FUNCTION_BLOCK UNIT_StateLogic (* Reduced PackML unit state machine: Reset/Start/Clear only from the occupation owner and only in a valid state; Execute runs the procedure until it reports DONE (Complete) or FAILED (Aborted) *)
  (* Standard: 61499-2 *)
  (* Version 0.1, 2026-09-28, Project contributors, AAU Smart Production Lab *)
  PACKAGE unitlib;
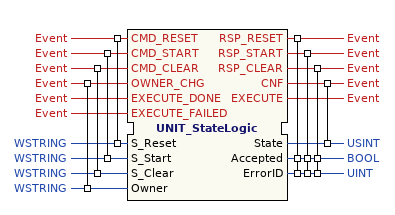
  EVENT_INPUT
    CMD_RESET WITH S_Reset;
    CMD_START WITH S_Start;
    CMD_CLEAR WITH S_Clear;
    OWNER_CHG WITH Owner;
    EXECUTE_DONE;
    EXECUTE_FAILED;
  END_EVENT
  EVENT_OUTPUT
    RSP_RESET WITH Accepted, ErrorID;
    RSP_START WITH Accepted, ErrorID;
    RSP_CLEAR WITH Accepted, ErrorID;
    CNF WITH State;
    EXECUTE;
  END_EVENT
  VAR_INPUT
    S_Reset : WSTRING;
    S_Start : WSTRING;
    S_Clear : WSTRING;
    Owner : WSTRING;
  END_VAR
  VAR_OUTPUT
    State : USINT := 2;
    Accepted : BOOL;
    ErrorID : UINT;
  END_VAR
  VAR
    Owned : BOOL;
  END_VAR
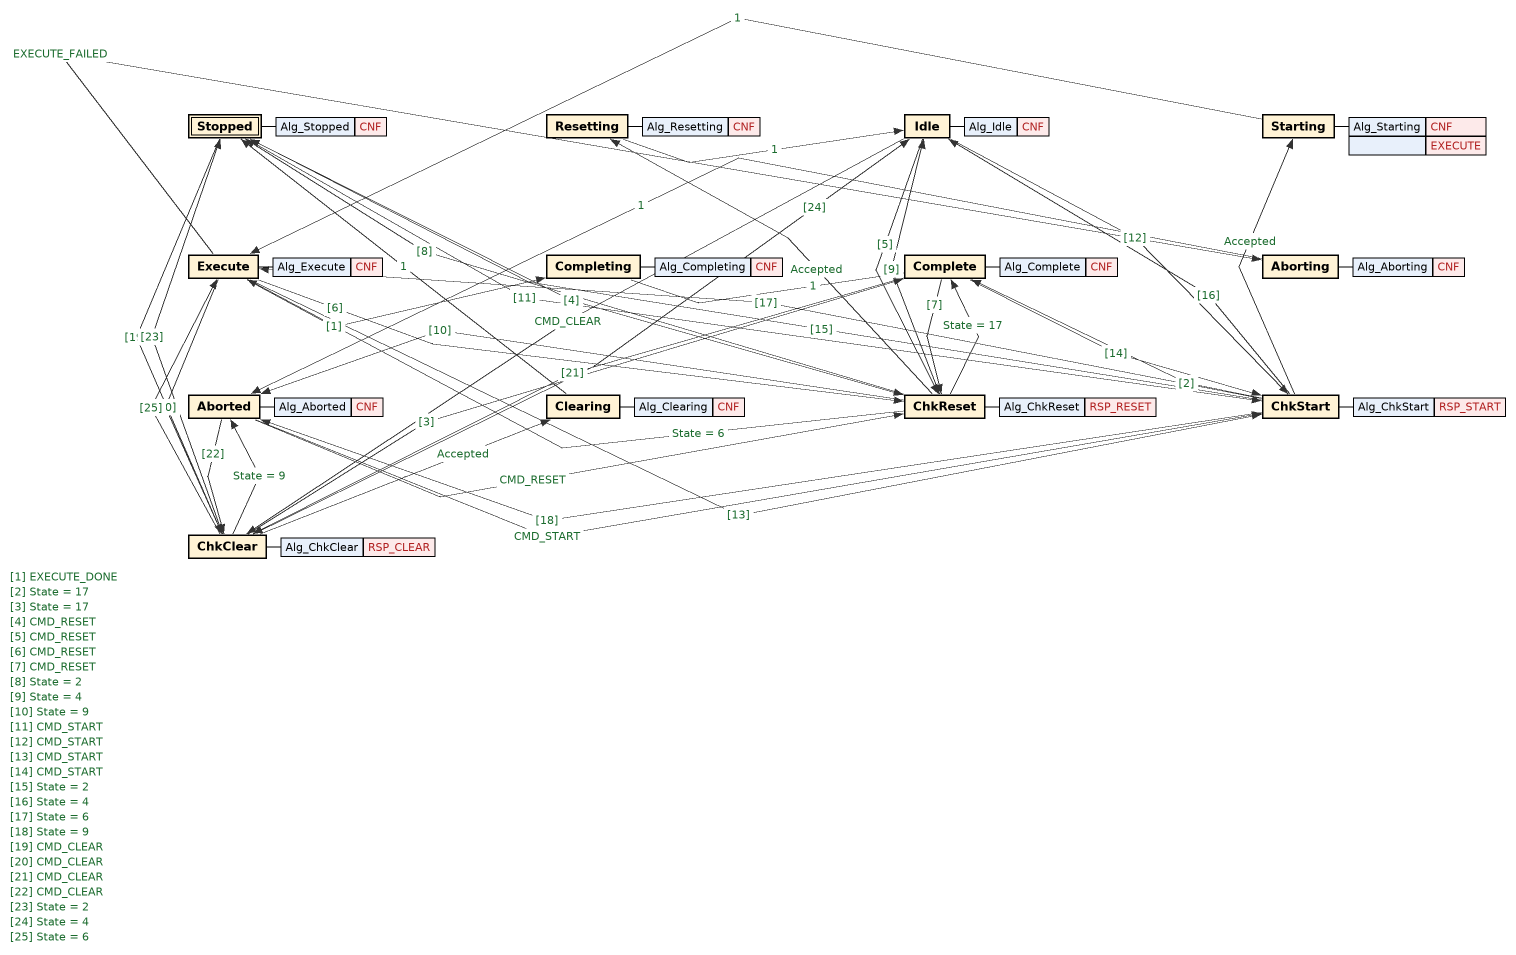
  EC_STATES
    Stopped : Alg_Stopped -> CNF;
    Resetting : Alg_Resetting -> CNF;
    Idle : Alg_Idle -> CNF;
    Starting : Alg_Starting -> CNF, -> EXECUTE;
    Execute : Alg_Execute -> CNF;
    Completing : Alg_Completing -> CNF;
    Complete : Alg_Complete -> CNF;
    Aborting : Alg_Aborting -> CNF;
    Aborted : Alg_Aborted -> CNF;
    Clearing : Alg_Clearing -> CNF;
    ChkReset : Alg_ChkReset -> RSP_RESET;
    ChkStart : Alg_ChkStart -> RSP_START;
    ChkClear : Alg_ChkClear -> RSP_CLEAR;
  END_STATES
  EC_TRANSITIONS
    Stopped TO ChkReset := CMD_RESET;
    Idle TO ChkReset := CMD_RESET;
    Execute TO ChkReset := CMD_RESET;
    Complete TO ChkReset := CMD_RESET;
    Aborted TO ChkReset := CMD_RESET;
    ChkReset TO Resetting := Accepted;
    ChkReset TO Stopped := State = 2;
    ChkReset TO Idle := State = 4;
    ChkReset TO Execute := State = 6;
    ChkReset TO Complete := State = 17;
    ChkReset TO Aborted := State = 9;
    Stopped TO ChkStart := CMD_START;
    Idle TO ChkStart := CMD_START;
    Execute TO ChkStart := CMD_START;
    Complete TO ChkStart := CMD_START;
    Aborted TO ChkStart := CMD_START;
    ChkStart TO Starting := Accepted;
    ChkStart TO Stopped := State = 2;
    ChkStart TO Idle := State = 4;
    ChkStart TO Execute := State = 6;
    ChkStart TO Complete := State = 17;
    ChkStart TO Aborted := State = 9;
    Stopped TO ChkClear := CMD_CLEAR;
    Idle TO ChkClear := CMD_CLEAR;
    Execute TO ChkClear := CMD_CLEAR;
    Complete TO ChkClear := CMD_CLEAR;
    Aborted TO ChkClear := CMD_CLEAR;
    ChkClear TO Clearing := Accepted;
    ChkClear TO Stopped := State = 2;
    ChkClear TO Idle := State = 4;
    ChkClear TO Execute := State = 6;
    ChkClear TO Complete := State = 17;
    ChkClear TO Aborted := State = 9;
    Resetting TO Idle := 1;
    Starting TO Execute := 1;
    Execute TO Completing := EXECUTE_DONE;
    Execute TO Aborting := EXECUTE_FAILED;
    Completing TO Complete := 1;
    Aborting TO Aborted := 1;
    Clearing TO Stopped := 1;
  END_TRANSITIONS
  ALGORITHM Alg_Stopped IN ST:
State := 2;
  END_ALGORITHM
  ALGORITHM Alg_Resetting IN ST:
State := 15;
  END_ALGORITHM
  ALGORITHM Alg_Idle IN ST:
State := 4;
  END_ALGORITHM
  ALGORITHM Alg_Starting IN ST:
State := 3;
  END_ALGORITHM
  ALGORITHM Alg_Execute IN ST:
State := 6;
  END_ALGORITHM
  ALGORITHM Alg_Completing IN ST:
State := 16;
  END_ALGORITHM
  ALGORITHM Alg_Complete IN ST:
State := 17;
  END_ALGORITHM
  ALGORITHM Alg_Aborting IN ST:
State := 8;
  END_ALGORITHM
  ALGORITHM Alg_Aborted IN ST:
State := 9;
  END_ALGORITHM
  ALGORITHM Alg_Clearing IN ST:
State := 1;
  END_ALGORITHM
  ALGORITHM Alg_ChkReset IN ST:
Owned := (S_Reset = Owner) AND (Owner <> "");
Accepted := Owned AND ((State = 2) OR (State = 17));
IF NOT Owned THEN
  ErrorID := 5;
ELSIF NOT Accepted THEN
  ErrorID := 4;
ELSE
  ErrorID := 0;
END_IF;
  END_ALGORITHM
  ALGORITHM Alg_ChkStart IN ST:
Owned := (S_Start = Owner) AND (Owner <> "");
Accepted := Owned AND ((State = 4));
IF NOT Owned THEN
  ErrorID := 5;
ELSIF NOT Accepted THEN
  ErrorID := 4;
ELSE
  ErrorID := 0;
END_IF;
  END_ALGORITHM
  ALGORITHM Alg_ChkClear IN ST:
Owned := (S_Clear = Owner) AND (Owner <> "");
Accepted := Owned AND ((State = 9));
IF NOT Owned THEN
  ErrorID := 5;
ELSIF NOT Accepted THEN
  ErrorID := 4;
ELSE
  ErrorID := 0;
END_IF;
  END_ALGORITHM
END_FUNCTION_BLOCK
